// TIA Portal V17 export
// export: Created 2025-06-26T07:49:14.4772247Z, ExportSetting WithDefaults, DisplayName Totally Integrated Automation Portal, DisplayVersion V17 Update 8, DisplayName TIA Portal Openness, DisplayVersion V17 Update 8, DisplayName TIA Portal Version Control Interface, DisplayVersion V17, DisplayName STEP 7 Professional, DisplayVersion V17 Update 8, DisplayName STEP 7 Safety, DisplayVersion V17 Update 6, DisplayName WinCC Advanced, DisplayVersion V17 Update 8
DATA_BLOCK "DB_Puma"   // DB7
{ S7_Optimized_Access := 'TRUE' }
VERSION : 0.1
// stored: AutoNumber true, DBAccessibleFromOPCUA true, IsOnlyStoredInLoadMemory false, IsRetainMemResEnabled false, IsWriteProtectedInAS false, MemoryReserve 100
   VAR
      Watchdog : "stHeartbeatCount2";   // Comm monitoring Puma <-> Heatbooster
      "CAN-Reset_Required" { S7_SetPoint := 'True'} : Bool;   // Manually reset the CAN comm
   END_VAR
BEGIN
   Watchdog.bEnable := true;
   Watchdog.tTimeout := T#2s;
END_DATA_BLOCK
